FUNCTION_BLOCK ARRAY2ARRAY_1440_LREAL (* Converter SIFB for LREAL arrays of length 96 *)
  (* Standard: 61499-2 *)
  (* Version 0.0, 2017-06-12, 4DIAC-IDE, 4DIAC-Consortium *)
  (* Version 1.0, 2017-06-12, Marc Jakobi, HTW Berlin *)
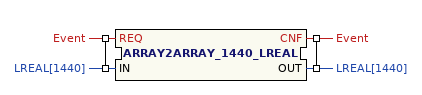
  EVENT_INPUT
    REQ WITH IN; (* Service Request *)
  END_EVENT
  EVENT_OUTPUT
    CNF WITH OUT; (* Confirmation of Requested Service *)
  END_EVENT
  VAR_INPUT
    IN : ARRAY [0..1439] OF LREAL; (* array input *)
  END_VAR
  VAR_OUTPUT
    OUT : ARRAY [0..1439] OF LREAL; (* array output *)
  END_VAR
  SERVICE APPLICATION/RESOURCE (* Converter SIFB for LREAL arrays of length 96 *)
    SEQUENCE request_inhibited
      APPLICATION.REQ-(SD) -> APPLICATION.CNF-(STATUS);
    END_SEQUENCE
  END_SERVICE
END_FUNCTION_BLOCK
